# B&R Automation Studio project DeboxPP70
Automation Studio 4.6.3.55 SP

## Configuration Config230524

CPU 4PPC70.0702-20B, AutomationRuntime B4.62, Build 4.1.2, Vc V4.62.0

### Task classes (Cpu.sw)
```
Cyclic#4:
  Robot <- Robot.prg
VcDataObjects: VisuRo <- VisuRobot.dob
```

### Hardware
```
4PPC70_0702_20B : 4PPC70.0702-20B v1.4.0.0
  Connector IF2:
    ActivateDevice = 1
    Mode = Manual
    InternetAddress = 10.16.7.34
    SubnetMask = 255.255.0.0
    Vnc1
    VncAuthentication1 = 1
    VncPasswordViewOnly1 = v
    VncRefreshRate1 = 100
  ConfigurationID = DeboxPP70_Config230524
  VcObjectName = VisuRo
  KeyMappingFile = VC\4PPC70_0702_20B.dis
staubli_io : FBE.staubli_io v1.0 (OrderNumber=staubli_io)  [PLK1 -> 4PPC70_0702_20B.IF1 [Cable Type=PowerlinkCable, Length=10, Version=1.0.0.2]]
  Supervision = off
```

### IoMap.iom - 4PPC70_0702_20B/IoMap.iom
```iecst
VAR_CONFIG
	::Robot:BOOL_Bouteille_1 AT %QX."staubli_io".POWERLINK_1_Q0Out;
END_VAR
```

## Logical view

### Program Logical/Robot (IEC)

#### Variables.var
```iecst
VAR
	BP_Bouteille_1 : BOOL;
	BOOL_Bouteille_1 : BOOL;
END_VAR
```

#### Main.st
```iecst
PROGRAM _INIT
END_PROGRAM

PROGRAM _CYCLIC
		(* Insert code here *)

	BOOL_Bouteille_1 := BP_Bouteille_1;

END_PROGRAM

END_PROGRAM

PROGRAM _EXIT
		(* Insert code here *)
END_PROGRAM
```

- Visualisation Logical/VisuRobot (not shown)

Listed in the project but not available here: Logical/Global.typ, Logical/Global.var, Logical/Libraries
